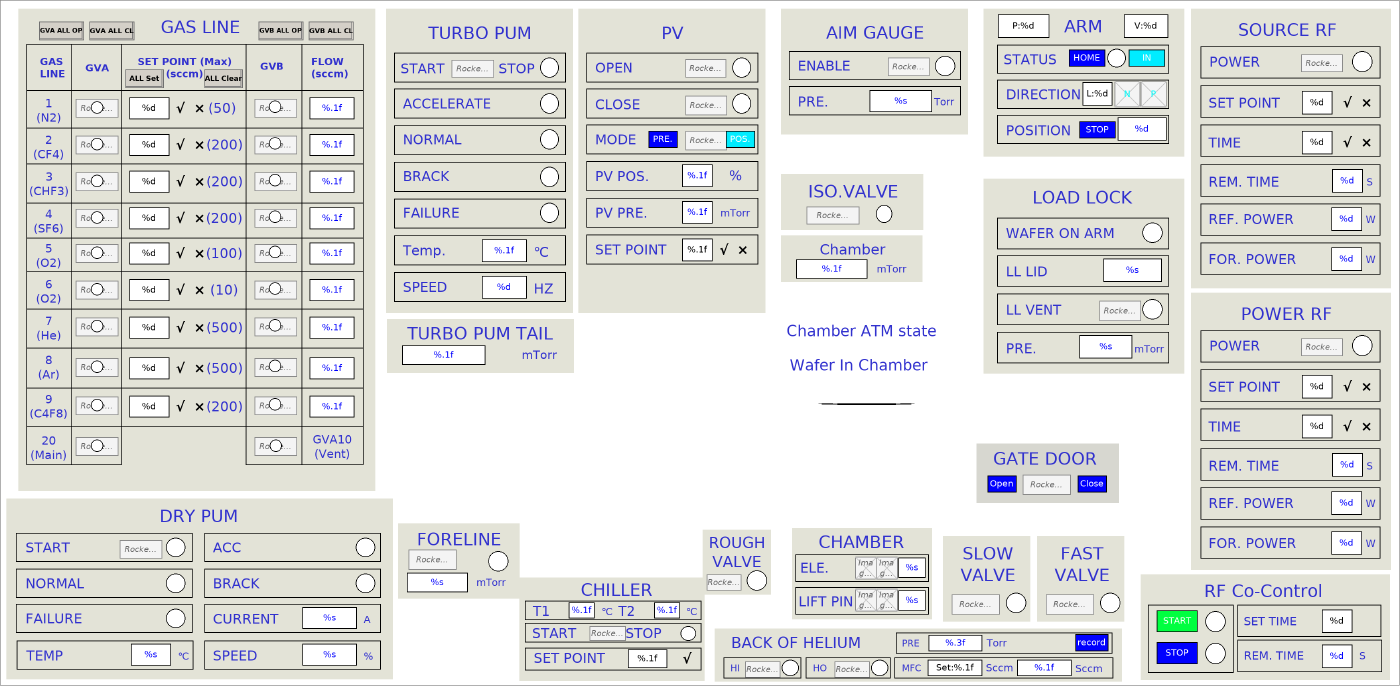
VISUALIZATION Overview  // 1755x860, background image ImagePool1.autoImg
    RoundedRectangle (23,11 447x604)
    RoundedRectangle (1233,11 251x185), colour toggle: NOT FuncModule_RS232_ARM.serialConnected, input disabled if: NOT FuncModule_RS232_ARM.serialConnected
    Label (1262,12 192x42), "ARM"
    RoundedRectangle (1250,56 215x36)
    RoundedRectangle (1250,100 215x36)
    Label (1258,108 110x21), "DIRECTION"
    RoundedRectangle (1250,144 215x36)
    Label (1258,153 96x21), "POSITION"
    RoundedRectangle (1340,62 45x21), "HOME", colour toggle: gICP.I_ARMHome, input disabled if: NOT FuncModule_RS232_ARM.serialConnected
        OnMouseClick: write the text variable via Default
        OnMouseClick: execute { gICP.ARM.Act_HOME(gICP.ARM.NoteHMI); }
    Label (1255,64 82x21), "STATUS"
    RoundedRectangle (1415,62 45x21), "IN", colour toggle: gICP.I_ARMHome or gICP.ARM.busy, input disabled if: NOT FuncModule_RS232_ARM.serialConnected
        OnMouseClick: write the text variable via Default
        OnMouseClick: execute { gICP.ARM.Act_IN(gICP.ARM.NoteHMI); }
    Ellipse (1388,61 23x23), colour toggle: gICP.ARM.busy or gICP.ARM.jogBusy
    Image (1397,102 32x32), "N", input disabled if: NOT FuncModule_RS232_ARM.serialConnected, image: VisuSymbols.Symbols.ArrowBoldLeft
        OnMouseClick: write the text variable via Default
        OnMouseClick: execute { gICP.ARM.Act_DirectionJog(_noteHMI:=gICP.ARM.NoteHMI,FALSE,gICp.ARM.setvel,gICP.ARM.jogsetlen); }
    Image (1430,102 32x32), "P", input disabled if: NOT FuncModule_RS232_ARM.serialConnected, image: VisuSymbols.Symbols.ArrowBoldRight
        OnMouseClick: write the text variable via Default
        OnMouseClick: execute { gICP.ARM.Act_DirectionJog(_noteHMI:=gICP.ARM.NoteHMI,TRUE,gICp.ARM.setvel,gICP.ARM.jogsetlen); }
    Group (993,662 175x114)
        RoundedRectangle (0,0 175x114)
        Label (19,2 136x31), "CHAMBER"
        RoundedRectangle (4,33 167x34)
        Label (7,40 59x20), "ELE."
        RoundedRectangle (4,74 167x34)
        Label (5,82 79x20), "LIFT PIN"
        Image (79,36 27x28), colour toggle: gICP.ElectrodeCyl.extend, image: ImagePool1.up
            OnMouseClick: write the text variable via Default
            OnMouseClick: execute { gICP.ElectrodeCyl.HMIItf.extend:=true; }
        Image (105,36 27x28), colour toggle: gICP.ElectrodeCyl.retract, image: ImagePool1.down
            OnMouseClick: write the text variable via Default
            OnMouseClick: execute { gICP.ElectrodeCyl.HMIItf.retract:=true; }
        Image (79,76 27x28), colour toggle: gICP.LiftPinCyl.extend, image: ImagePool1.up
            OnMouseClick: write the text variable via Default
            OnMouseClick: execute { gICP.LiftPinCyl.HMIItf.extend:=true; }
        Image (105,76 27x28), colour toggle: gICP.LiftPinCyl.retract, image: ImagePool1.down
            OnMouseClick: write the text variable via Default
            OnMouseClick: execute { gICP.LiftPinCyl.HMIItf.retract:=true; }
        RoundedRectangle (133,37 34x25), "%s", text variable: gICP.ElectrodeCyl.HMIItf.sensorShow
        RoundedRectangle (133,78 34x25), "%s", text variable: gICP.LiftPinCyl.HMIItf.sensorShow
    Line (33,55) (455,55)
    Line (33,582) (152,582)
    Line (33,113) (455,113)
    Line (33,160) (455,160)
    Line (33,205) (455,205)
    Line (33,254) (455,254)
    Line (33,298) (455,298)
    Line (33,340) (455,340)
    Line (33,387) (455,387)
    Line (33,486) (455,486)
    Line (33,55) (33,582)
    Line (89,55) (89,582)
    Line (152,55) (152,582)
    Line (308,55) (308,582)
    Line (378,55) (378,582)
    Line (455,55) (455,582)
    Label (40,13 423x42), "GAS LINE"
    Label (47,61 45x48), "GAS LINE"
    Label (104,61 42x48), "GVA"
    Label (387,61 59x48), "FLOW (sccm)"
    Label (323,59 45x48), "GVB"
    Label (168,61 127x48), "SET POINT (Max) (sccm)"
    RockerSwitch (95,124 53x23), variable: gICP.GVA1Valve.HMIItf.singleControl, behaviour: TOGGLE, style: Switch-RockerSwitch-Blue
    RockerSwitch (95,170 53x23), variable: gICP.GVA2Valve.HMIItf.singleControl, behaviour: TOGGLE, style: Switch-RockerSwitch-Blue
    RockerSwitch (95,216 53x23), variable: gICP.GVA3Valve.HMIItf.singleControl, behaviour: TOGGLE, style: Switch-RockerSwitch-Blue
    RockerSwitch (95,262 53x23), variable: gICP.GVA4Valve.HMIItf.singleControl, behaviour: TOGGLE, style: Switch-RockerSwitch-Blue
    RockerSwitch (95,306 53x23), variable: gICP.GVA5Valve.HMIItf.singleControl, behaviour: TOGGLE, style: Switch-RockerSwitch-Blue
    RockerSwitch (95,352 53x23), variable: gICP.GVA6Valve.HMIItf.singleControl, behaviour: TOGGLE, style: Switch-RockerSwitch-Blue
    RockerSwitch (95,449 53x23), variable: gICP.GVA8Valve.HMIItf.singleControl, behaviour: TOGGLE, style: Switch-RockerSwitch-Blue
    RockerSwitch (95,548 53x23), variable: gICP.GV20Valve_Main.HMIItf.singleControl, behaviour: TOGGLE, style: Switch-RockerSwitch-Blue
    RockerSwitch (319,124 53x23), variable: gICP.GVB1Valve.HMIItf.singleControl, behaviour: TOGGLE, style: Switch-RockerSwitch-Blue
    RockerSwitch (319,170 53x23), variable: gICP.GVB2Valve.HMIItf.singleControl, behaviour: TOGGLE, style: Switch-RockerSwitch-Blue
    RockerSwitch (319,216 53x23), variable: gICP.GVB3Valve.HMIItf.singleControl, behaviour: TOGGLE, style: Switch-RockerSwitch-Blue
    RockerSwitch (319,262 53x23), variable: gICP.GVB4Valve.HMIItf.singleControl, behaviour: TOGGLE, style: Switch-RockerSwitch-Blue
    RockerSwitch (319,306 53x23), variable: gICP.GVB5Valve.HMIItf.singleControl, behaviour: TOGGLE, style: Switch-RockerSwitch-Blue
    RockerSwitch (319,352 53x23), variable: gICP.GVB6Valve.HMIItf.singleControl, behaviour: TOGGLE, style: Switch-RockerSwitch-Blue
    RockerSwitch (319,449 53x23), variable: gICP.GVB8Valve.HMIItf.singleControl, behaviour: TOGGLE, style: Switch-RockerSwitch-Blue
    RoundedRectangle (388,448 56x27), "%.1f", text variable: gICP.MFC8.actflowFloat, colour toggle: NOT FuncModule_RS485_MFC.serialConnected
    RoundedRectangle (388,350 56x27), "%.1f", text variable: gICP.MFC6.actflowFloat, colour toggle: NOT FuncModule_RS485_MFC.serialConnected
    RoundedRectangle (388,304 56x27), "%.1f", text variable: gICP.MFC5.actflowFloat, colour toggle: NOT FuncModule_RS485_MFC.serialConnected
    RoundedRectangle (388,260 56x27), "%.1f", text variable: gICP.MFC4.actflowFloat, colour toggle: NOT FuncModule_RS485_MFC.serialConnected
    RoundedRectangle (388,214 56x27), "%.1f", text variable: gICP.MFC3.actflowFloat, colour toggle: NOT FuncModule_RS485_MFC.serialConnected
    RoundedRectangle (388,168 56x27), "%.1f", text variable: gICP.MFC2.actflowFloat, colour toggle: NOT FuncModule_RS485_MFC.serialConnected
    RoundedRectangle (388,122 56x27), "%.1f", text variable: gICP.MFC1.actflowFloat, colour toggle: NOT FuncModule_RS485_MFC.serialConnected
    Rectangle (162,122 50x27), "%d", text variable: gICP.MFC1.setFlow, colour toggle: gICP.MFC1.setdone
        OnMouseClick: write the text variable via Default
    Rectangle (215,122 23x27), "√", colour toggle: gICP.MFC1.setbusy
        OnMouseClick: write the text variable via Default
        OnMouseClick: execute { gICP.MFC1.MFCHMItif.set:=TRUE; }
    Rectangle (241,122 18x27), "×", colour toggle: gICP.MFC1.clearbusy
        OnMouseClick: write the text variable via Default
        OnMouseClick: execute { gICP.MFC1.MFCHMItif.clear:=TRUE; }
    Label (259,126 39x19), "(50)"
    Rectangle (162,168 50x27), "%d", text variable: gICP.MFC2.setFlow, colour toggle: gICP.MFC2.setdone
        OnMouseClick: write the text variable via Default
    Rectangle (215,168 23x27), "√", colour toggle: gICP.MFC2.setbusy
        OnMouseClick: write the text variable via Default
        OnMouseClick: execute { gICP.MFC2.MFCHMItif.set:=TRUE; }
    Rectangle (241,168 18x27), "×", colour toggle: gICP.MFC2.clearbusy
        OnMouseClick: write the text variable via Default
        OnMouseClick: execute { gICP.MFC2.MFCHMItif.clear:=TRUE; }
    Label (259,172 45x19), "(200)"
    Rectangle (162,214 50x27), "%d", text variable: gICP.MFC3.setFlow, colour toggle: gICP.MFC3.setdone
        OnMouseClick: write the text variable via Default
    Rectangle (215,214 23x27), "√", colour toggle: gICP.MFC3.setbusy
        OnMouseClick: write the text variable via Default
        OnMouseClick: execute { gICP.MFC3.MFCHMItif.set:=TRUE; }
    Rectangle (241,214 18x27), "×", colour toggle: gICP.MFC3.clearbusy
        OnMouseClick: write the text variable via Default
        OnMouseClick: execute { gICP.MFC3.MFCHMItif.clear:=TRUE; }
    Label (259,218 45x19), "(200)"
    Rectangle (162,260 50x27), "%d", text variable: gICP.MFC4.setFlow, colour toggle: gICP.MFC4.setdone
        OnMouseClick: write the text variable via Default
    Rectangle (215,260 23x27), "√", colour toggle: gICP.MFC4.setbusy
        OnMouseClick: write the text variable via Default
        OnMouseClick: execute { gICP.MFC4.MFCHMItif.set:=TRUE; }
    Rectangle (241,260 18x27), "×", colour toggle: gICP.MFC4.clearbusy
        OnMouseClick: write the text variable via Default
        OnMouseClick: execute { gICP.MFC4.MFCHMItif.clear:=TRUE; }
    Label (259,264 44x19), "(200)"
    Rectangle (162,304 50x27), "%d", text variable: gICP.MFC5.setFlow, colour toggle: gICP.MFC5.setdone
        OnMouseClick: write the text variable via Default
    Rectangle (215,304 23x27), "√", colour toggle: gICP.MFC5.setbusy
        OnMouseClick: write the text variable via Default
        OnMouseClick: execute { gICP.MFC5.MFCHMItif.set:=TRUE; }
    Rectangle (241,304 18x27), "×", colour toggle: gICP.MFC5.clearbusy
        OnMouseClick: write the text variable via Default
        OnMouseClick: execute { gICP.MFC5.MFCHMItif.clear:=TRUE; }
    Label (259,308 44x19), "(100)"
    Rectangle (162,350 50x27), "%d", text variable: gICP.MFC6.setFlow, colour toggle: gICP.MFC6.setdone
        OnMouseClick: write the text variable via Default
    Rectangle (215,350 23x27), "√", colour toggle: gICP.MFC6.setbusy
        OnMouseClick: write the text variable via Default
        OnMouseClick: execute { gICP.MFC6.MFCHMItif.set:=TRUE; }
    Rectangle (241,350 18x27), "×", colour toggle: gICP.MFC6.clearbusy
        OnMouseClick: write the text variable via Default
        OnMouseClick: execute { gICP.MFC6.MFCHMItif.clear:=TRUE; }
    Label (259,354 44x19), "(10)"
    Rectangle (162,448 50x27), "%d", text variable: gICP.MFC8.setFlow, colour toggle: gICP.MFC8.setdone
        OnMouseClick: write the text variable via Default
    Rectangle (215,448 23x27), "√", colour toggle: gICP.MFC8.setbusy
        OnMouseClick: write the text variable via Default
        OnMouseClick: execute { gICP.MFC8.MFCHMItif.set:=TRUE; }
    Rectangle (241,448 18x27), "×", colour toggle: gICP.MFC8.clearbusy
        OnMouseClick: write the text variable via Default
        OnMouseClick: execute { gICP.MFC8.MFCHMItif.clear:=TRUE; }
    Label (259,452 45x19), "(500)"
    Label (39,116 44x45), "1 (N2)"
    Label (39,162 44x45), "2 (CF4)"
    Label (39,255 44x45), "4 (SF6)"
    Label (35,208 53x45), "3 (CHF3)"
    Label (39,343 44x45), "6 (O2)"
    Label (39,298 44x45), "5 (O2)"
    Label (39,539 44x45), "20 (Main)"
    Label (39,438 44x45), "8 (Ar)"
    Ellipse (114,127 15x15), colour toggle: gICP.GVA1Valve.extRelay
    Ellipse (114,173 15x15), colour toggle: gICP.GVA2Valve.extRelay
    Ellipse (114,219 15x15), colour toggle: gICP.GVA3Valve.extRelay
    Ellipse (114,265 15x15), colour toggle: gICP.GVA4Valve.extRelay
    Ellipse (114,309 15x15), colour toggle: gICP.GVA5Valve.extRelay
    Ellipse (114,355 15x15), colour toggle: gICP.GVA6Valve.extRelay
    Ellipse (114,452 15x15), colour toggle: gICP.GVA8Valve.extRelay
    Ellipse (114,551 15x15), colour toggle: gICP.GV20Valve_Main.extRelay
    Ellipse (337,126 15x15), colour toggle: gICP.GVB1Valve.extRelay
    Ellipse (337,172 15x15), colour toggle: gICP.GVB2Valve.extRelay
    Ellipse (337,218 15x15), colour toggle: gICP.GVB3Valve.extRelay
    Ellipse (337,264 15x15), colour toggle: gICP.GVB4Valve.extRelay
    Ellipse (337,308 15x15), colour toggle: gICP.GVB5Valve.extRelay
    Ellipse (337,354 15x15), colour toggle: gICP.GVB6Valve.extRelay
    Ellipse (337,451 15x15), colour toggle: gICP.GVB8Valve.extRelay
    Line (33,534) (455,534)
    RockerSwitch (95,497 53x23), variable: gICP.GVA9Valve.HMIItf.singleControl, behaviour: TOGGLE, style: Switch-RockerSwitch-Blue
    RockerSwitch (319,497 53x23), variable: gICP.GVB9Valve.HMIItf.singleControl, behaviour: TOGGLE, style: Switch-RockerSwitch-Blue
    RoundedRectangle (388,496 56x27), "%.1f", text variable: gICP.MFC9.actflowFloat, colour toggle: NOT FuncModule_RS485_MFC.serialConnected
    Rectangle (162,496 50x27), "%d", text variable: gICP.MFC9.setFlow, colour toggle: gICP.MFC9.setdone
        OnMouseClick: write the text variable via Default
    Rectangle (215,496 23x27), "√", colour toggle: gICP.MFC9.setbusy
        OnMouseClick: write the text variable via Default
        OnMouseClick: execute { gICP.MFC9.MFCHMItif.set:=TRUE; }
    Rectangle (241,496 18x27), "×", colour toggle: gICP.MFC9.clearbusy
        OnMouseClick: write the text variable via Default
        OnMouseClick: execute { gICP.MFC9.MFCHMItif.clear:=TRUE; }
    Label (259,500 45x19), "(200)"
    Label (36,487 50x45), "9 (C4F8)"
    Ellipse (114,500 15x15), colour toggle: gICP.GVA9Valve.extRelay
    Ellipse (337,499 15x15), colour toggle: gICP.GVB9Valve.extRelay
    Line (33,436) (455,436)
    RockerSwitch (95,398 53x23), variable: gICP.GVA7Valve.HMIItf.singleControl, behaviour: TOGGLE, style: Switch-RockerSwitch-Blue
    RockerSwitch (319,398 53x23), variable: gICP.GVB7Valve.HMIItf.singleControl, behaviour: TOGGLE, style: Switch-RockerSwitch-Blue
    RoundedRectangle (388,397 56x27), "%.1f", text variable: gICP.MFC7.actflowFloat, colour toggle: NOT FuncModule_RS485_MFC.serialConnected
    Rectangle (162,397 50x27), "%d", text variable: gICP.MFC7.setFlow, colour toggle: gICP.MFC7.setdone
        OnMouseClick: write the text variable via Default
    Rectangle (215,397 23x27), "√", colour toggle: gICP.MFC7.setbusy
        OnMouseClick: write the text variable via Default
        OnMouseClick: execute { gICP.MFC7.MFCHMItif.set:=TRUE; }
    Rectangle (241,397 18x27), "×", colour toggle: gICP.MFC7.clearbusy
        OnMouseClick: write the text variable via Default
        OnMouseClick: execute { gICP.MFC7.MFCHMItif.clear:=TRUE; }
    Label (259,401 45x19), "(500)"
    Label (39,389 44x45), "7 (He)"
    Ellipse (114,401 15x15), colour toggle: gICP.GVA7Valve.extRelay
    Ellipse (337,400 15x15), colour toggle: gICP.GVB7Valve.extRelay
    Rectangle (92,118 55x31)
        tap gICP.GVA1Valve.HMIItf.singleControltemp
    Rectangle (92,164 55x31)
        tap gICP.GVA2Valve.HMIItf.singleControltemp
    Rectangle (92,211 55x31)
        tap gICP.GVA3Valve.HMIItf.singleControltemp
    Rectangle (92,258 55x31)
        tap gICP.GVA4Valve.HMIItf.singleControltemp
    Rectangle (92,300 55x31)
        tap gICP.GVA5Valve.HMIItf.singleControltemp
    Rectangle (92,346 55x31)
        tap gICP.GVA6Valve.HMIItf.singleControltemp
    Rectangle (92,392 55x31)
        tap gICP.GVA7Valve.HMIItf.singleControltemp
    Rectangle (92,442 55x31)
        tap gICP.GVA8Valve.HMIItf.singleControltemp
    Rectangle (92,492 55x31)
        tap gICP.GVA9Valve.HMIItf.singleControltemp
    Rectangle (92,543 55x31)
        tap gICP.GV20Valve_Main.HMIItf.singleControltemp
    Rectangle (316,119 55x31)
        tap gICP.GVB1Valve.HMIItf.singleControltemp
    Rectangle (316,165 55x31)
        tap gICP.GVB2Valve.HMIItf.singleControltemp
    Rectangle (316,212 55x31)
        tap gICP.GVB3Valve.HMIItf.singleControltemp
    Rectangle (316,257 55x31)
        tap gICP.GVB4Valve.HMIItf.singleControltemp
    Rectangle (316,301 55x31)
        tap gICP.GVB5Valve.HMIItf.singleControltemp
    Rectangle (316,347 55x31)
        tap gICP.GVB6Valve.HMIItf.singleControltemp
    Rectangle (316,393 55x31)
        tap gICP.GVB7Valve.HMIItf.singleControltemp
    Rectangle (316,443 55x31)
        tap gICP.GVB8Valve.HMIItf.singleControltemp
    Rectangle (316,491 55x31)
        tap gICP.GVB9Valve.HMIItf.singleControltemp
    RoundedRectangle (725,11 234x381), colour toggle: gICP.PDV.error
    Label (747,20 192x43), "PV"
    RoundedRectangle (735,66 215x37)
    RockerSwitch (859,74 51x23), variable: gICP.PDV.HMIItf.open, behaviour: TOGGLE, style: Switch-RockerSwitch-Blue
    Ellipse (918,72 23x25), colour toggle: gICP.PDVOpenSensor
    Label (743,74 117x22), "OPEN"
    RoundedRectangle (735,111 215x37)
    RockerSwitch (859,120 52x24), variable: gICP.PDV.HMIItf.close, behaviour: TOGGLE, style: Switch-RockerSwitch-Blue
    Ellipse (918,117 23x25), colour toggle: gICP.PDVCloseSensor
    Label (743,120 117x22), "CLOSE"
    RoundedRectangle (735,156 215x37)
    Label (743,164 69x22), "MODE"
    RoundedRectangle (735,202 215x37)
    Label (743,210 87x22), "PV POS."
    RoundedRectangle (735,248 215x37)
    Label (743,256 87x22), "PV PRE."
    RoundedRectangle (735,294 215x37)
    Label (743,302 106x22), "SET POINT"
    Rectangle (855,299 38x28), "%.1f", text variable: gICP.PDV.HMIItf.setPressure, colour toggle: gICP.PDV.HMIItf.setPointNotEq, input disabled if: gICP.PDV.error
        OnMouseClick: write the text variable via Default
    RockerSwitch (859,164 52x24), variable: gICP.PDV.HMIItf.mode, behaviour: TOGGLE, style: Switch-RockerSwitch-Blue
    RoundedRectangle (813,164 36x21), "PRE.", colour toggle: gICP.PDVModeRelay
    RoundedRectangle (910,164 36x21), "POS.", colour toggle: gICP.PDVModeRelay
    Label (911,209 23x22), "%"
    RoundedRectangle (855,206 38x28), "%.1f", text variable: gICP.PDV.actPos
    RoundedRectangle (855,252 38x28), "%.1f", text variable: gICP.PDV.actPressure
    Label (900,256 47x22), "mTorr"
    Rectangle (897,299 22x28), "√", colour toggle: gICP.PDV.HMIItf.setflag, input disabled if: gICP.PDV.error
        OnMouseClick: write the text variable via Default
        OnMouseClick: execute { gICP.PDV.HMIItf.set:=true; }
    Rectangle (922,299 18x28), "×", colour toggle: gICP.PDV.HMIItf.clearflag, input disabled if: gICP.PDV.error
        OnMouseClick: write the text variable via Default
        OnMouseClick: execute { gICP.PDV.HMIItf.clear:=true; }
    Rectangle (857,158 55x30), input disabled if: gICP.PDV.error
        tap gICP.PDV.HMIItf.modetemp
    Rectangle (857,115 55x31)
        tap gICP.PDV.HMIItf.closetemp
    Rectangle (852,69 62x30)
        tap gICP.PDV.HMIItf.opentemp
    RoundedRectangle (484,11 234x381), colour toggle: Not FuncModule_RS232_TBP.serialConnected
    Label (506,20 192x43), "TURBO PUM"
    RoundedRectangle (494,66 215x37)
    Ellipse (677,72 23x25), colour toggle: gICP.TruboPumOpen
    Label (499,75 67x22), "START"
    RoundedRectangle (494,111 215x37)
    RoundedRectangle (494,203 215x37)
    Ellipse (677,162 23x25), colour toggle: gICP.TruboPumNormal
    Label (502,164 117x22), "NORMAL"
    RoundedRectangle (494,157 215x37)
    Ellipse (677,117 23x25), colour toggle: gICP.TruboPumAcc
    Label (502,119 140x22), "ACCELERATE"
    RoundedRectangle (494,249 215x37)
    Ellipse (677,209 23x25), colour toggle: gICP.TruboPumDcc
    Label (502,210 117x22), "BRACK"
    RoundedRectangle (494,295 215x37)
    Ellipse (677,254 23x25), colour toggle: gICP.TruboPumError
    Label (502,256 117x22), "FAILURE"
    RoundedRectangle (494,341 215x37)
    Label (502,349 70x22), "SPEED"
    Label (666,351 31x22), "HZ"
    RoundedRectangle (604,346 56x28), "%d", text variable: gICP.TruboPumRotationSpeed
    Label (622,75 57x22), "STOP"
    RockerSwitch (566,75 53x22), variable: gICP.TruboPum.HMIItf.singleControl, behaviour: TOGGLE, style: Switch-RockerSwitch-Blue
    Label (502,303 105x22), "Temp."
    Label (666,305 31x22), "℃"
    RoundedRectangle (604,300 56x28), "%.1f", text variable: gICP.TruboPumTMS
    Rectangle (564,70 55x31)
        tap gICP.TruboPum.HMIItf.singleControltemp
    RoundedRectangle (651,724 232x129)
    RoundedRectangle (658,781 221x24)
    Label (692,728 162x23), "CHILLER"
    RoundedRectangle (658,753 221x24)
    Label (665,758 49x16), "T1"
    RoundedRectangle (713,755 32x20), "%.1f", text variable: gICP.Chiller.RTD1, colour toggle: gICP.Chiller.Error
    Label (751,759 14x15), "℃"
    RockerSwitch (739,785 45x18), variable: gICP.Chiller.HMIItf.singleControl, behaviour: TOGGLE, style: Switch-RockerSwitch-Blue
    Ellipse (853,785 19x18), colour toggle: gICP.Chiller.extRelay
    Label (664,785 70x18), "START"
    Label (781,785 59x18), "STOP"
    RoundedRectangle (658,812 221x28)
    Label (666,816 89x18), "SET POINT"
    Rectangle (787,814 49x23), "%.1f", text variable: gICP.Chiller.setpointVal
        OnMouseClick: write the text variable via Default
    Rectangle (852,814 19x23), "√", colour toggle: gICP.Chiller.busy and gICP.Chiller.setStep<>0
        OnMouseClick: write the text variable via Default
        OnMouseClick: execute { gICP.Chiller.HMIItf.set:=TRUE; }
    Label (857,759 14x15), "℃"
    Label (772,758 49x16), "T2"
    RoundedRectangle (820,755 32x20), "%.1f", text variable: gICP.Chiller.RTD2, colour toggle: gICP.Chiller.Error
    Rectangle (734,780 52x26)
        tap gICP.Chiller.HMIItf.singleControltemp
    Group (8,625 484x226), input disabled if: gWarmShowHMI.showFlag
        RoundedRectangle (0,0 484x226)
        Label (30,1 423x42), "DRY PUM"
        RoundedRectangle (12,43 221x36)
        Ellipse (200,49 24x24), colour toggle: gICP.MachianicalPumOpen
        Label (21,51 172x21), "START"
        RoundedRectangle (248,43 221x36)
        Label (256,51 77x21), "ACC"
        RoundedRectangle (248,178 221x36)
        Label (256,186 97x22), "SPEED"
        Ellipse (438,49 24x24), colour toggle: gICP.MachianicalPum.Accing
        RockerSwitch (142,52 53x23), variable: gICP.MachianicalPum.HMIItf.singleControl, behaviour: TOGGLE, style: Switch-RockerSwitch-Blue
        RoundedRectangle (371,182 68x27), "%s", text variable: gICP.MachianicalPum.DryPumpSpeed
        Label (445,187 21x21), "%"
        RoundedRectangle (13,178 221x36)
        Label (22,186 134x22), "TEMP"
        RoundedRectangle (156,182 50x27), "%s", text variable: gICP.MachianicalPum.DryPumpTemperature
        Label (212,187 21x21), "℃"
        RoundedRectangle (12,88 221x36)
        Ellipse (200,94 24x24), colour toggle: gICP.MachianicalPum.Normal
        Label (21,96 100x21), "NORMAL"
        RoundedRectangle (248,88 221x36)
        Label (256,96 77x21), "BRACK"
        Ellipse (438,94 24x24), colour toggle: gICP.MachianicalPum.Dccing
        RoundedRectangle (12,132 221x36)
        Ellipse (200,138 24x24), colour toggle: gICP.MachianicalPumAlm
        Label (21,140 172x21), "FAILURE"
        RoundedRectangle (248,132 221x36)
        Label (256,140 97x22), "CURRENT"
        RoundedRectangle (371,136 68x27), "%s", text variable: gICP.MachianicalPum.DryPumpCurrent
        Label (445,141 21x21), "A"
        Rectangle (135,45 62x31)
            tap gICP.MachianicalPum.HMIItf.singleControltemp
    RoundedRectangle (499,656 152x94)
    Label (510,659 131x34), "FORELINE"
    RockerSwitch (512,689 60x25), variable: gICP.ForlinLineValve.HMIItf.singleControl, behaviour: TOGGLE, style: Switch-RockerSwitch-Blue
    Ellipse (612,691 25x25), colour toggle: gICP.ForlinLineValveExtRelay
    Label (594,719 50x22), "mTorr"
    RoundedRectangle (510,718 76x24), "%s", text variable: gICP.ForeLineGauge.outputValue_String, colour toggle: gICP.ForeLineGauge.error
    Rectangle (508,684 68x31)
        tap gICP.ForlinLineValve.HMIItf.singleControltemp
    RoundedRectangle (979,218 178x70)
    Label (981,226 177x28), "ISO.VALVE"
    RockerSwitch (1011,259 66x22), variable: gICP.ISOValve.HMIItf.singleControl, behaviour: TOGGLE, style: Switch-RockerSwitch-Blue
    Ellipse (1098,257 20x22), colour toggle: gICP.ISOExtRelay
    Rectangle (1011,255 60x27)
        tap gICP.ISOValve.HMIItf.singleControltemp
    Group (1233,224 251x244), input disabled if: gWarmShowHMI.showFlag
        RoundedRectangle (0,0 251x244)
        Label (24,1 199x45), "LOAD LOCK"
        RoundedRectangle (17,49 215x39)
        Ellipse (199,55 25x25), colour toggle: gICP.I_WaferCheck
        Label (25,57 167x23), "WAFER ON ARM"
        RoundedRectangle (17,96 215x39)
        Label (25,105 117x23), "LL LID"
        RoundedRectangle (17,192 215x39)
        Label (25,201 94x24), "PRE."
        RoundedRectangle (17,144 215x39)
        Ellipse (199,151 25x25), colour toggle: gICP.VentExtRelay
        Label (25,153 140x23), "LL VENT"
        RoundedRectangle (150,100 73x29), "%s", text variable: gICP.I_LLSwitchString
        RockerSwitch (145,153 52x25), variable: gICP.VentValve.HMIItf.singleControl, behaviour: TOGGLE, style: Switch-RockerSwitch-Blue
        RoundedRectangle (120,196 66x29), "%s", text variable: gICP.LoadLockGauge.outputValue_String, colour toggle: gICP.LoadLockGauge.error
        Label (186,202 48x23), "mTorr"
        Rectangle (137,146 60x31)
            tap gICP.VentValve.HMIItf.singleControltemp
    Group (1224,556 178x74), input disabled if: gWarmShowHMI.showFlag
        RoundedRectangle (0,0 178x74)
        Label (5,3 162x32), "GATE DOOR"
        RockerSwitch (58,39 60x25), variable: gICP.GateDoorValve.HMIItf.singleControl, behaviour: TOGGLE, style: Switch-RockerSwitch-Blue
        RoundedRectangle (127,40 36x21), "Close", colour toggle: gICP.GateDoorRetSensor
        RoundedRectangle (14,40 36x21), "Open", colour toggle: gICP.GateDoorExtSensor
        Rectangle (55,34 65x31)
            tap gICP.GateDoorValve.HMIItf.singleControltemp
    Group (1182,672 227x107), input disabled if: gWarmShowHMI.showFlag
        RoundedRectangle (118,0 109x107)
        Label (128,4 93x63), "FAST VALVE"
        RockerSwitch (129,73 60x25), variable: gICP.FastPummingValve.HMIItf.singleControl, behaviour: TOGGLE, style: Switch-RockerSwitch-Blue
        Ellipse (197,71 25x25), colour toggle: gICP.FastPummingExtRelay
        RoundedRectangle (0,0 109x107)
        Label (10,4 93x63), "SLOW VALVE"
        RockerSwitch (11,73 60x25), variable: gICP.SlowPummingValve.HMIItf.singleControl, behaviour: TOGGLE, style: Switch-RockerSwitch-Blue
        Ellipse (79,71 25x25), colour toggle: gICP.SlowPummingExtRelay
        Rectangle (8,69 65x31)
            tap gICP.SlowPummingValve.HMIItf.singleControltemp
        Rectangle (126,69 65x31)
            tap gICP.FastPummingValve.HMIItf.singleControltemp
    RoundedRectangle (1493,367 250x347), colour toggle: gICP.PowerRF.error
    Label (1517,370 192x47), "POWER RF"
    RoundedRectangle (1505,414 225x40)
    RockerSwitch (1631,424 52x22), variable: gICP.PowerRF.openRelay, behaviour: TOGGLE, style: Switch-RockerSwitch-Blue
    Ellipse (1695,420 25x26), colour toggle: gICP.PowerRFOpenRelay
    Label (1513,422 117x23), "POWER"
    RoundedRectangle (1505,562 225x40)
    RoundedRectangle (1505,611 225x40)
    RoundedRectangle (1505,660 225x40)
    RoundedRectangle (1505,463 225x40)
    Label (1512,474 111x22), "SET POINT"
    Rectangle (1632,470 38x29), "%d", text variable: gICP.PowerRF.HMIItf.setpower, colour toggle: gICP.PowerRF.HMIItf.setpower<>gICP.PowerRF.setpower or gICP.PowerRF.setpower<>gICP.PowerRF.setpowerRead, input disabled if: S_CO_ControlRF.busy
        OnMouseClick: write the text variable via Default
    Rectangle (1678,470 23x29), "√", input disabled if: S_CO_ControlRF.busy
        OnMouseClick: write the text variable via Default
        OnMouseClick: execute { gICP.PowerRF.setpower:=gICP.PowerRF.HMIItf.setpower; gICP.PowerRF.Act_Write(); }
    Rectangle (1704,470 18x29), "×", input disabled if: S_CO_ControlRF.busy
        OnMouseClick: write the text variable via Default
        OnMouseClick: execute {
            gICP.PowerRF.setpower:=0;
            gICP.PowerRF.HMIItf.setpower:=0;
            gICP.PowerRF.Act_Write();
        }
    RoundedRectangle (1505,512 225x40)
    Label (1512,524 111x22), "TIME"
    Rectangle (1632,520 38x29), "%d", text variable: gICP.PowerRF.HMIItf.settime, colour toggle: gICP.PowerRF.HMIItf.settime<>gICP.PowerRF.settime
        OnMouseClick: write the text variable via Default
    Rectangle (1678,520 23x29), "√"
        OnMouseClick: write the text variable via Default
        OnMouseClick: execute { gICP.PowerRF.settime:=gICP.PowerRF.HMIItf.settime; }
    Rectangle (1704,520 18x29), "×"
        OnMouseClick: write the text variable via Default
        OnMouseClick: execute { gICP.PowerRF.settime:=0; gICP.PowerRF.HMIItf.settime:=0; }
    Label (1512,573 155x22), "REM. TIME"
    RoundedRectangle (1670,568 38x29), "%d", text variable: gICP.PowerRF.rematime, colour toggle: gICP.PowerRF.rematime<>0
    Label (1710,573 16x22), "S"
    Label (1512,620 155x22), "REF. POWER"
    RoundedRectangle (1669,616 38x29), "%d", text variable: gICP.PowerRF.reflectedpower, colour toggle: gICP.PowerRF.reflectedpower<>0
    Label (1709,620 16x22), "W"
    Label (1512,670 155x22), "FOR. POWER"
    RoundedRectangle (1669,666 38x29), "%d", text variable: gICP.PowerRF.forwardpower, colour toggle: (gICP.PowerRF.openbusy AND ABS(gICP.PowerRF.forwardpower-gICP.PowerRF.setpower)>2) OR (not gICP.PowerRF.busy and gICP.PowerRF.forwardpower>0) OR (gICP.PowerRF.closebusy and gICP.PowerRF.forwardpower>0)
    Label (1709,670 16x22), "W"
    Rectangle (1624,419 65x31), input disabled if: S_CO_ControlRF.busy
        tap gICP.PowerRF.HMIItf.singleControltemp
    RoundedRectangle (979,11 234x157)
    Label (1001,20 192x42), "AIM GAUGE"
    RoundedRectangle (989,64 215x36)
    RockerSwitch (1113,72 52x23), variable: gICP.AIMValve.HMIItf.singleControl, behaviour: TOGGLE, style: Switch-RockerSwitch-Blue
    Ellipse (1172,70 25x25), colour toggle: gICP .AIMExtRelay
    Label (997,72 117x21), "ENABLE"
    RoundedRectangle (989,108 215x36)
    Label (997,117 90x21), "PRE."
    RoundedRectangle (1090,113 78x27), "%s", text variable: gICP.AIMGauge.outputValue_String, colour toggle: gICP.AIMGauge.error
    Label (1168,117 34x21), "Torr"
    Rectangle (1106,66 65x31)
        tap gICP.AIMValve.HMIItf.singleControltemp
    RoundedRectangle (881,664 85x81)
    Label (883,668 82x49), "ROUGH VALVE"
    RockerSwitch (886,720 43x20), variable: gICP.RoughValve.HMIItf.singleControl, behaviour: TOGGLE, style: Switch-RockerSwitch-Blue
    Ellipse (936,715 25x25), colour toggle: gICP.RoughValveExtRelay
    Rectangle (882,714 52x26)
        tap gICP.RoughValve.HMIItf.singleControltemp
    Button (49,27 56x23), "GVA ALL OP", colour toggle: gICP.S_GASBOX_AllGVAOpen
        tap gICP.C_GASBOX_AllGVAOpenTemp
    Button (112,27 56x23), "GVA ALL CL", colour toggle: gICP.S_GASBOX_AllGVAClose
        tap gICP.C_GASBOX_AllGVACloseTemp
    Button (387,27 56x23), "GVB ALL CL", colour toggle: gICP.S_GASBOX_AllGVBClose
        tap gICP.C_GASBOX_AllGVBCloseTemp
    Button (324,27 56x23), "GVB ALL OP", colour toggle: gICP.S_GASBOX_AllGVBOpen
        tap gICP.C_GASBOX_AllGVBOpenTemp
    Button (157,87 48x23), "ALL Set"
        tap gICP.C_GASBOX_AllMFCSetTemp
    Button (256,87 48x23), "ALL Clear"
        tap gICP.C_GASBOX_AllMFCClearTemp
    RoundedRectangle (1493,11 250x350), colour toggle: gICP.SourceRF.error
    Label (1518,14 192x47), "SOURCE RF"
    RoundedRectangle (1505,58 225x40)
    RockerSwitch (1631,68 52x22), variable: gICP.SourceRF.openRelay, behaviour: TOGGLE, style: Switch-RockerSwitch-Blue
    Ellipse (1695,64 25x26), colour toggle: gICP.SourceRFOpenRelay
    Label (1513,66 117x23), "POWER"
    RoundedRectangle (1505,206 225x40)
    RoundedRectangle (1505,255 225x40)
    RoundedRectangle (1505,304 225x40)
    RoundedRectangle (1505,107 225x40)
    Label (1512,118 111x22), "SET POINT"
    Rectangle (1632,114 38x29), "%d", text variable: gICP.SourceRF.HMIItf.setpower, colour toggle: gICP.SourceRF.HMIItf.setpower<>gICP.SourceRF.setpower or gICP.SourceRF.setpower<>gICP.SourceRF.setpowerRead, input disabled if: S_CO_ControlRF.busy
        OnMouseClick: write the text variable via Default
    Rectangle (1678,114 23x29), "√", input disabled if: S_CO_ControlRF.busy
        OnMouseClick: write the text variable via Default
        OnMouseClick: execute { gICP.SourceRF.setpower:=gICP.SourceRF.HMIItf.setpower; gICP.SourceRF.Act_Write(); }
    Rectangle (1704,114 18x29), "×", input disabled if: S_CO_ControlRF.busy
        OnMouseClick: write the text variable via Default
        OnMouseClick: execute {
            gICP.SourceRF.setpower:=0;
            gICP.SourceRF.HMIItf.setpower:=0;
            gICP.SourceRF.Act_Write();
        }
    RoundedRectangle (1505,156 225x40)
    Label (1512,168 111x22), "TIME"
    Rectangle (1632,164 38x29), "%d", text variable: gICP.SourceRF.HMIItf.settime, colour toggle: gICP.SourceRF.HMIItf.settime<>gICP.SourceRF.settime
        OnMouseClick: write the text variable via Default
    Rectangle (1678,164 23x29), "√"
        OnMouseClick: write the text variable via Default
        OnMouseClick: execute { gICP.SourceRF.settime:=gICP.SourceRF.HMIItf.settime; }
    Rectangle (1704,164 18x29), "×"
        OnMouseClick: write the text variable via Default
        OnMouseClick: execute { gICP.SourceRF.settime:=0; gICP.SourceRF.HMIItf.settime:=0; }
    Label (1512,217 155x22), "REM. TIME"
    RoundedRectangle (1670,212 38x29), "%d", text variable: gICP.SourceRF.rematime, colour toggle: gICP.SourceRF.rematime<>0
    Label (1710,217 16x22), "S"
    Label (1512,264 155x22), "REF. POWER"
    RoundedRectangle (1669,260 38x29), "%d", text variable: gICP.SourceRF.reflectedpower, colour toggle: gICP.SourceRF.reflectedpower<>0
    Label (1709,264 16x22), "W"
    Label (1512,314 155x22), "FOR. POWER"
    RoundedRectangle (1669,310 38x29), "%d", text variable: gICP.SourceRF.forwardpower, colour toggle: (gICP.SourceRF.openbusy AND ABS(gICP.SourceRF.forwardpower-gICP.SourceRF.setpower)>2) OR (not gICP.SourceRF.busy and gICP.SourceRF.forwardpower>0)
    Label (1709,314 16x22), "W"
    Rectangle (1623,63 65x31), input disabled if: S_CO_ControlRF.busy
        tap gICP.SourceRF.HMIItf.singleControltemp
    RoundedRectangle (1401,147 61x29), "%d", text variable: gICP.ARM.actpos
    Rectangle (1251,18 64x29), "P:%d", text variable: gARMPosition
        OnMouseClick: write the text variable via Default, min 0, max 9000
    Rectangle (1409,18 55x29), "V:%d", text variable: gICP.ARM.setvel
        OnMouseClick: write the text variable via Default, min 1, max 30
    Rectangle (1357,103 37x29), "L:%d", text variable: gICP.ARM.jogsetlen
        OnMouseClick: write the text variable via Default, min 1, max 10
    RoundedRectangle (1353,152 45x21), "STOP", input disabled if: NOT FuncModule_RS232_ARM.serialConnected
        OnMouseClick: write the text variable via Default
        OnMouseClick: execute { gICP.ARM.Act_Stop(); }
    Line (308,582) (455,582)
    Label (386,539 61x42), "GVA10 (Vent)"
    RockerSwitch (319,548 53x23), variable: gICP.GVA10Valve_Vent.HMIItf.singleControl, behaviour: TOGGLE, style: Switch-RockerSwitch-Blue
    Ellipse (338,551 15x15), colour toggle: gICP.GVA10Valve_Vent.extRelay
    Rectangle (316,543 55x31)
        tap gICP.GVA10Valve_Vent.HMIItf.singleControltemp
    RoundedRectangle (1430,720 312x132)
    Label (1488,723 192x36), "RF Co-Control"
    RoundedRectangle (1551,802 181x40)
    Label (1556,811 97x22), "REM. TIME"
    RoundedRectangle (1657,808 38x29), "%d", text variable: gCO_ControlRFRMTime, colour toggle: gCO_ControlRFRMTime>1
    Label (1701,811 16x22), "S"
    RoundedRectangle (1551,758 180x40)
    Label (1556,768 96x22), "SET TIME"
    Rectangle (1657,764 38x29), "%d", text variable: gCO_ControlRFTime
        OnMouseClick: write the text variable via Default
    RoundedRectangle (1439,758 107x85)
    RoundedRectangle (1450,765 51x27), "START", input disabled if: NOT(gICP.PowerRF.openCondition AND gICP.SourceRF.openCondition) OR S_CO_ControlRF.busy
        OnMouseClick: write the text variable via Default
        OnMouseClick: execute {
            S_CO_ControlRF.Act_Init_Status();
            S_CO_ControlRF.Act_Ex();
            S_CO_ControlRF.bTrig:=TRUE;
        }
    Ellipse (1511,766 25x26), colour toggle: S_CO_ControlRF.busy
    RoundedRectangle (1450,805 51x27), "STOP"
        OnMouseClick: write the text variable via Default
        OnMouseClick: execute { S_CO_ControlRF.bStop:=TRUE; S_CO_ControlRF.bAbort:=TRUE; }
    Ellipse (1511,806 25x26), colour toggle: S_CO_ControlRF.stopDone
    Rectangle (896,791 52x26)
        tap gICP.RoughValve.HMIItf.singleControltemp
    RoundedRectangle (896,788 510x66)
    Label (905,789 186x34), "BACK OF HELIUM"
    RoundedRectangle (907,824 97x26)
    RockerSwitch (934,829 44x20), variable: gICP.HeINValve.HMIItf.singleControl, behaviour: TOGGLE, style: Switch-RockerSwitch-Blue
    Ellipse (980,827 21x20), colour toggle: gICP.HeINExtRelay
    Label (909,827 25x21), "HI"
    RoundedRectangle (1010,824 106x26)
    RockerSwitch (1046,829 44x20), variable: gICP.HePumValve.HMIItf.singleControl, behaviour: TOGGLE, style: Switch-RockerSwitch-Blue
    Ellipse (1092,827 21x20), colour toggle: gICP.HePumExtRelay
    Label (1012,827 32x21), "HO"
    RoundedRectangle (1123,793 271x26)
    Label (1126,796 32x21), "PRE"
    RoundedRectangle (1121,824 274x26)
    Label (1127,827 32x21), "MFC"
    Label (1234,795 41x22), "Torr"
    RoundedRectangle (1164,796 67x20), "%.3f", text variable: gICP.HeCheckGaugeReal
    RoundedRectangle (1275,827 68x20), "%.1f", text variable: gICP.HeMFC_ActFlow
    Label (1345,827 44x22), "Sccm"
    Rectangle (934,824 41x26)
        tap gICP.HeINValve.HMIItf.singleControltemp
    Rectangle (1046,824 41x26)
        tap gICP.HePumValve.HMIItf.singleControltemp
    Ellipse (1026,505 120x2), colour toggle: gWaferMemoryState=1
        OnMouseClick: execute { gWaferMemoryState:=BOOL_TO_INT(NOT INT_TO_BOOL(gWaferMemoryState)); ups_CX51X0.Act_Wrtie(); }
    Label (988,442 177x32), "Wafer In Chamber", invisible if: NOT otherMachineState.lightShow
    Label (965,399 230x32), "Chamber ATM state", invisible if: NOT gICP.I_ATMSensor
    RoundedRectangle (979,295 177x58)
    Label (994,300 150x26), "Chamber"
    Label (1096,326 50x22), "mTorr"
    RoundedRectangle (998,325 89x24), "%.1f", text variable: gICP.ChamberGauge.outputValue1, colour toggle: gICP.ChamberGauge.error
    Rectangle (1163,827 68x20), "Set:%.1f", text variable: gICP.HeMFC_SetFlowHMI
        OnMouseClick: write the text variable via Default, min 0, max 100
    Label (1233,826 41x22), "Sccm"
    RoundedRectangle (485,400 234x67)
    Label (496,405 212x26), "TURBO PUM TAIL"
    Label (651,434 50x22), "mTorr"
    RoundedRectangle (504,433 104x24), "%.1f", text variable: gICP.TBGauge.outputValue, colour toggle: gICP.TBGauge.error
    RoundedRectangle (1348,795 41x21), "record", colour toggle: MainRunPOU.testLog
        toggle MainRunPOU.testLog
        OnMouseClick: write the text variable via Default
END_VISUALIZATION

(* stored: Version 1.1.0.1, ProductVersion 3.1.4024.12
   Visu Overview: Id {9ca16f32-27d0-4d5b-b04b-9a30f3e54125} *)
